FUNCTION_BLOCK Model_HMI (* Service Interface Function Block Type *)
  (* Standard: 61499-2 *)
  (* Version 0.0, 5/29/2016, Andrei, nxtControl GmbH, template *)
  PACKAGE Main;
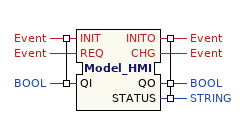
  EVENT_INPUT
    INIT WITH QI;
    REQ;
  END_EVENT
  EVENT_OUTPUT
    INITO WITH QO, STATUS;
    CHG;
  END_EVENT
  VAR_INPUT
    QI : BOOL;
  END_VAR
  VAR_OUTPUT
    QO : BOOL; (* Event Output Qualifier *)
    STATUS : STRING; (* Service Status *)
  END_VAR
  SERVICE /
    SEQUENCE 
    END_SEQUENCE
  END_SERVICE
END_FUNCTION_BLOCK
